INTERFACE I_CYLINDER_DA_TESTDEV1 EXTENDS I_CYLINDER_DA_TESTDEV2_4

METHOD M_LowPressureCalibration : BOOL
END_METHOD

METHOD M_LowPressureMode : BOOL
VAR_INPUT
  bSet:                            BOOL;
	ePressureType:                   E_PRESSURE_TYPE;
  rWorkPressure:                   REAL;
END_VAR
END_METHOD

METHOD M_OpenReservoir : BOOL
VAR_INPUT
  bOpenA:       BOOL;
  bOpenB:       BOOL;
END_VAR
END_METHOD

METHOD M_Pump2Add : BOOL
VAR_INPUT
  bAdd:         BOOL;
END_VAR
END_METHOD

METHOD M_Pump3Add : BOOL
VAR_INPUT
  bAdd:         BOOL;
END_VAR
END_METHOD

METHOD M_Pump4Add : BOOL
VAR_INPUT
  bAdd:         BOOL;
END_VAR
END_METHOD

PROPERTY P_ActiveVolumeFlow : REAL
GET
END_GET
END_PROPERTY

{warning 'Eigenschaftenimplementierung hinzufügen'}
PROPERTY P_CurrentLowPressureForceInN : REAL
GET
END_GET
END_PROPERTY

PROPERTY P_LowPressure : REAL
GET
END_GET
END_PROPERTY

PROPERTY P_LowPressureChA : REAL
GET
END_GET
END_PROPERTY

PROPERTY P_LowPressureChB : REAL
GET
END_GET
END_PROPERTY

PROPERTY P_LowPressureModeEnable : BOOL
GET
END_GET
END_PROPERTY

PROPERTY P_Pump2Added : BOOL
GET
END_GET
END_PROPERTY

PROPERTY P_Pump3Added : BOOL
GET
END_GET
END_PROPERTY

PROPERTY P_Pump4Added : BOOL
GET
END_GET
END_PROPERTY

PROPERTY P_ReservoirAOpened : BOOL
GET
END_GET
END_PROPERTY

PROPERTY P_ReservoirBOpened : BOOL
GET
END_GET
END_PROPERTY

PROPERTY P_ReservoirPressure : REAL
GET
END_GET
END_PROPERTY

END_INTERFACE

(* stored: Version 1.1.0.1, ProductVersion 3.1.4024.12
   Itf I_CYLINDER_DA_TESTDEV1: Id {0198e8f2-4230-4629-be52-a2fb000ee511}
   Method M_LowPressureCalibration: Id {2da68073-ce8a-43b2-a453-452850389d9c}
   Method M_LowPressureMode: Id {43dea638-8c38-4ac4-b13e-1eb9b149f543}
   Method M_OpenReservoir: Id {b3c674f5-535d-4bbd-a699-05a8457d80ba}
   Method M_Pump2Add: Id {6f1abf68-27be-4148-ad29-c6754ccfebb7}
   Method M_Pump3Add: Id {159a842f-9c46-475b-ae63-0d9a8d367968}
   Method M_Pump4Add: Id {178ca3c9-b10a-4aa9-a456-3453723144fa}
   Property P_ActiveVolumeFlow: Id {fa4f44bf-e9ae-4762-95d1-9395ca058a3c}
   Get Get: Id {22811cd3-2cf0-4de8-a67f-cdcbbd8409a2}
   Property P_CurrentLowPressureForceInN: Id {5e2b2c64-35c9-423a-ab4c-e5c1337e4d8d}
   Get Get: Id {4ba0715f-eb60-41ce-bcb7-0dcb241875f2}
   Property P_LowPressure: Id {60eaa627-61b2-4dad-8819-5f6ffa137b5e}
   Get Get: Id {3744e1d0-0b5e-4245-b4ac-dd2d21e7db05}
   Property P_LowPressureChA: Id {211fc384-59fc-4010-8712-d6217bb40880}
   Get Get: Id {c98939e9-33d8-4957-8140-d1e185e6340c}
   Property P_LowPressureChB: Id {6b79b5ad-707f-4a31-8f6c-6c9458a18b47}
   Get Get: Id {6cd434ed-6506-4304-bc91-421be317b57c}
   Property P_LowPressureModeEnable: Id {f59294a8-aee3-4792-9aca-6d780b5b9faf}
   Get Get: Id {64b7a803-da23-42a2-a593-004810120e1a}
   Property P_Pump2Added: Id {84cefa24-1313-4220-8466-c245a18911f4}
   Get Get: Id {c14ebfd1-1c9f-4d07-ab73-4ff8108c456d}
   Property P_Pump3Added: Id {73e2da8e-1558-4655-82c6-e3053c4f85b2}
   Get Get: Id {72e54fe6-c3b9-43f8-a69a-a272f6c101b3}
   Property P_Pump4Added: Id {26d15a5a-2ed8-4046-9331-dfc1fa11a485}
   Get Get: Id {d1de188b-ac79-47bd-8c98-c42ed0b4be00}
   Property P_ReservoirAOpened: Id {24f59d45-993d-4e13-baa0-effe55fb23ec}
   Get Get: Id {e15e2fb5-15a9-446e-b2f2-1a16a5db45f0}
   Property P_ReservoirBOpened: Id {f2b72622-f3ae-4e41-9f63-46403b4329fa}
   Get Get: Id {cf24a253-5371-4aaa-9b91-42faeda0f6b0}
   Property P_ReservoirPressure: Id {158f0d06-f5ad-4362-bb47-dd438d93fe81}
   Get Get: Id {728aaab0-aee3-4fc4-b52f-73a16ab5e19c} *)
